(* Logix 5000 project; controller CLASE_1 Emulate 5570 rev 28.11; software revision 28.02; part 14 of 15 *)
(* tags used below, declared in another part *)
   FV_00_Intlk_Ok : BOOL;
   FV_00_Perm_Ok : BOOL;
   P_100_B_Intlk_OK : BOOL;
   PID_OUT_TK_200 : REAL;   // Esfuerzo de control Deberá ir direccionada a la salida analogica fisica
   PID_OUT_TK_300 : REAL;
   PPX_M_100 : P_DescList[1];
   PPX_M_200 : P_DescList[1];
   PPX_M_300 : P_DescList[1];
   PPX_P_100_B : P_DescList[1];
   PPX_P_200 : P_DescList[1];
   PPX_P_300 : P_DescList[1];
   PPX_Pump_100_A : P_DescList[1];
   Pump_100_A_Intlk_Ok : BOOL;

PROGRAM Equipos_TK_100   (* main routine MainProgram *)
VAR
   P_51A_B_Perm : P_Perm := (Inp_Perm01 := 1, Inp_Perm02 := 1, Inp_Perm03 := 1, Inp_Perm04 := 1, Inp_Perm05 := 1, Inp_Perm06 := 1, Inp_Perm07 := 1, Inp_Perm08 := 1, Inp_Perm09 := 1, Inp_Perm10 := 1, Inp_Perm11 := 1, Inp_Perm12 := 1, Inp_Perm13 := 1, Inp_Perm14 := 1, Inp_Perm15 := 1, Cfg_OKState := 2#1111_1111_1111_1111, Sts_Perm := 2#1111_1111_1111_1110);
   P_AIn_01 : P_AIn := (Inp_HiHiGate := 1, Inp_HiGate := 1, Inp_LoGate := 1, Inp_LoLoGate := 1, Inp_FailGate := 1, Cfg_SetTrack := 1, Cfg_PCmdClear := 1, Cfg_HiHiAckReqd := 1, Cfg_HiAckReqd := 1, Cfg_LoAckReqd := 1, Cfg_LoLoAckReqd := 1, Cfg_FailAckReqd := 1, Cfg_HiHiSeverity := 750, Cfg_HiSeverity := 500, Cfg_LoSeverity := 500, Cfg_LoLoSeverity := 750, Cfg_FailSeverity := 1000, Cfg_InpRawMax := 100.0, Cfg_PVEUMax := 100.0, Cfg_HiHiDB := 1.0, Cfg_HiDB := 1.0, Cfg_LoDB := 1.0, Cfg_LoLoDB := 1.0, Cfg_FailHiLim := 103.958336, Cfg_FailLoLim := -2.0833333, Cfg_FailDB := 0.41666666, PSet_HiHiLim := 1.5e+38, PSet_HiLim := 1.5e+38, PSet_LoLim := -1.5e+38, PSet_LoLoLim := -1.5e+38, OSet_HiHiLim := 1.5e+38, OSet_HiLim := 1.5e+38, OSet_LoLim := -1.5e+38, OSet_LoLoLim := -1.5e+38, Val_PVMinCapt := 1.5e+38, Val_PVMaxCapt := -1.5e+38, Val_PVEUMax := 100.0, Val_HiHiLim := 1.5e+38, Val_HiLim := 1.5e+38, Val_LoLim := -1.5e+38, Val_LoLoLim := -1.5e+38, Sts_InpPV := 1, Sts_Oper := 1, Ack_HiHi := 1, Ack_Hi := 1, Ack_Lo := 1, Ack_LoLo := 1, Ack_Fail := 1);
   P_AIn_02 : P_AIn := (Inp_HiHiGate := 1, Inp_HiGate := 1, Inp_LoGate := 1, Inp_LoLoGate := 1, Inp_FailGate := 1, Cfg_SetTrack := 1, Cfg_PCmdClear := 1, Cfg_HiHiAckReqd := 1, Cfg_HiAckReqd := 1, Cfg_LoAckReqd := 1, Cfg_LoLoAckReqd := 1, Cfg_FailAckReqd := 1, Cfg_HiHiSeverity := 750, Cfg_HiSeverity := 500, Cfg_LoSeverity := 500, Cfg_LoLoSeverity := 750, Cfg_FailSeverity := 1000, Cfg_InpRawMax := 100.0, Cfg_PVEUMax := 100.0, Cfg_HiHiDB := 1.0, Cfg_HiDB := 1.0, Cfg_LoDB := 1.0, Cfg_LoLoDB := 1.0, Cfg_FailHiLim := 103.958336, Cfg_FailLoLim := -2.0833333, Cfg_FailDB := 0.41666666, PSet_HiHiLim := 1.5e+38, PSet_HiLim := 1.5e+38, PSet_LoLim := -1.5e+38, PSet_LoLoLim := -1.5e+38, OSet_HiHiLim := 1.5e+38, OSet_HiLim := 1.5e+38, OSet_LoLim := -1.5e+38, OSet_LoLoLim := -1.5e+38, Val_PVMinCapt := 1.5e+38, Val_PVMaxCapt := -1.5e+38, Val_PVEUMax := 100.0, Val_HiHiLim := 1.5e+38, Val_HiLim := 1.5e+38, Val_LoLim := -1.5e+38, Val_LoLoLim := -1.5e+38, Sts_InpPV := 1, Sts_Oper := 1, Ack_HiHi := 1, Ack_Hi := 1, Ack_Lo := 1, Ack_LoLo := 1, Ack_Fail := 1);
   P_AIn_03 : P_AIn := (Inp_HiHiGate := 1, Inp_HiGate := 1, Inp_LoGate := 1, Inp_LoLoGate := 1, Inp_FailGate := 1, Cfg_SetTrack := 1, Cfg_PCmdClear := 1, Cfg_HiHiAckReqd := 1, Cfg_HiAckReqd := 1, Cfg_LoAckReqd := 1, Cfg_LoLoAckReqd := 1, Cfg_FailAckReqd := 1, Cfg_HiHiSeverity := 750, Cfg_HiSeverity := 500, Cfg_LoSeverity := 500, Cfg_LoLoSeverity := 750, Cfg_FailSeverity := 1000, Cfg_InpRawMax := 100.0, Cfg_PVEUMax := 100.0, Cfg_HiHiDB := 1.0, Cfg_HiDB := 1.0, Cfg_LoDB := 1.0, Cfg_LoLoDB := 1.0, Cfg_FailHiLim := 103.958336, Cfg_FailLoLim := -2.0833333, Cfg_FailDB := 0.41666666, PSet_HiHiLim := 1.5e+38, PSet_HiLim := 1.5e+38, PSet_LoLim := -1.5e+38, PSet_LoLoLim := -1.5e+38, OSet_HiHiLim := 1.5e+38, OSet_HiLim := 1.5e+38, OSet_LoLim := -1.5e+38, OSet_LoLoLim := -1.5e+38, Val_PVMinCapt := 1.5e+38, Val_PVMaxCapt := -1.5e+38, Val_PVEUMax := 100.0, Val_HiHiLim := 1.5e+38, Val_HiLim := 1.5e+38, Val_LoLim := -1.5e+38, Val_LoLoLim := -1.5e+38, Sts_InpPV := 1, Sts_Oper := 1, Ack_HiHi := 1, Ack_Hi := 1, Ack_Lo := 1, Ack_LoLo := 1, Ack_Fail := 1);
   P_AIn_04 : P_AIn := (Inp_HiHiGate := 1, Inp_HiGate := 1, Inp_LoGate := 1, Inp_LoLoGate := 1, Inp_FailGate := 1, Cfg_SetTrack := 1, Cfg_PCmdClear := 1, Cfg_HiHiAckReqd := 1, Cfg_HiAckReqd := 1, Cfg_LoAckReqd := 1, Cfg_LoLoAckReqd := 1, Cfg_FailAckReqd := 1, Cfg_HiHiSeverity := 750, Cfg_HiSeverity := 500, Cfg_LoSeverity := 500, Cfg_LoLoSeverity := 750, Cfg_FailSeverity := 1000, Cfg_InpRawMax := 100.0, Cfg_PVEUMax := 100.0, Cfg_HiHiDB := 1.0, Cfg_HiDB := 1.0, Cfg_LoDB := 1.0, Cfg_LoLoDB := 1.0, Cfg_FailHiLim := 103.958336, Cfg_FailLoLim := -2.0833333, Cfg_FailDB := 0.41666666, PSet_HiHiLim := 1.5e+38, PSet_HiLim := 1.5e+38, PSet_LoLim := -1.5e+38, PSet_LoLoLim := -1.5e+38, OSet_HiHiLim := 1.5e+38, OSet_HiLim := 1.5e+38, OSet_LoLim := -1.5e+38, OSet_LoLoLim := -1.5e+38, Val_PVMinCapt := 1.5e+38, Val_PVMaxCapt := -1.5e+38, Val_PVEUMax := 100.0, Val_HiHiLim := 1.5e+38, Val_HiLim := 1.5e+38, Val_LoLim := -1.5e+38, Val_LoLoLim := -1.5e+38, Sts_InpPV := 1, Sts_Oper := 1, Ack_HiHi := 1, Ack_Hi := 1, Ack_Lo := 1, Ack_LoLo := 1, Ack_Fail := 1);
   P_DIn_01 : P_DIn := (Inp_PV := 1, Inp_Target := 1, Inp_Gate := 1, Cfg_NormTextVis := 1, Cfg_PCmdClear := 1, Cfg_TgtDisagreeAckReqd := 1, Cfg_TgtDisagreeSeverity := 750, Ack_TgtDisagree := 1);
   P_DIn_02 : P_DIn := (Inp_PV := 1, Inp_Target := 1, Inp_Gate := 1, Cfg_NormTextVis := 1, Cfg_PCmdClear := 1, Cfg_TgtDisagreeAckReqd := 1, Cfg_TgtDisagreeSeverity := 750, Ack_TgtDisagree := 1);
   P_DIn_03 : P_DIn := (Inp_PV := 1, Inp_Target := 1, Inp_Gate := 1, Cfg_NormTextVis := 1, Cfg_PCmdClear := 1, Cfg_TgtDisagreeAckReqd := 1, Cfg_TgtDisagreeSeverity := 750, Ack_TgtDisagree := 1);
   P_Intlk_01 : P_Intlk := (Cfg_PCmdClear := 1, Sts_IntlkOK := 1, Sts_NBIntlkOK := 1);
   P_Intlk_02 : P_Intlk := (Cfg_PCmdClear := 1, Sts_IntlkOK := 1, Sts_NBIntlkOK := 1);
   P_Intlk_03 : P_Intlk := (Cfg_PCmdClear := 1, Sts_IntlkOK := 1, Sts_NBIntlkOK := 1);
   P_Intlk_04 : P_Intlk := (Cfg_PCmdClear := 1, Sts_IntlkOK := 1, Sts_NBIntlkOK := 1);
   P_Intlk_05 : P_Intlk := (Cfg_PCmdClear := 1, Sts_IntlkOK := 1, Sts_NBIntlkOK := 1);
   P_Intlk_06 : P_Intlk := (Cfg_PCmdClear := 1, Sts_IntlkOK := 1, Sts_NBIntlkOK := 1);
   P_Motor_01 : P_Motor := (Inp_PermOK := 1, Inp_NBPermOK := 1, Inp_IntlkOK := 1, Inp_NBIntlkOK := 1, Cfg_PCmdClear := 1, Cfg_ShedOnFailToStart := 1, Cfg_ShedOnIOFault := 1, Cfg_FailToStartAckReqd := 1, Cfg_FailToStopAckReqd := 1, Cfg_IntlkTripAckReqd := 1, Cfg_IOFaultAckReqd := 1, Cfg_FailToStartSeverity := 1000, Cfg_FailToStopSeverity := 1000, Cfg_IntlkTripSeverity := 500, Cfg_IOFaultSeverity := 1000, Cfg_SimFdbkT := 2, Cfg_FailToStartT := 10, Cfg_FailToStopT := 10, Sts_Stopped := 1, Sts_Oper := 1, Ack_FailToStart := 1, Ack_FailToStop := 1, Ack_IntlkTrip := 1, Ack_IOFault := 1);
   P_Motor_02 : P_Motor := (Inp_PermOK := 1, Inp_NBPermOK := 1, Inp_IntlkOK := 1, Inp_NBIntlkOK := 1, Cfg_PCmdClear := 1, Cfg_ShedOnFailToStart := 1, Cfg_ShedOnIOFault := 1, Cfg_FailToStartAckReqd := 1, Cfg_FailToStopAckReqd := 1, Cfg_IntlkTripAckReqd := 1, Cfg_IOFaultAckReqd := 1, Cfg_FailToStartSeverity := 1000, Cfg_FailToStopSeverity := 1000, Cfg_IntlkTripSeverity := 500, Cfg_IOFaultSeverity := 1000, Cfg_SimFdbkT := 2, Cfg_FailToStartT := 10, Cfg_FailToStopT := 10, Sts_Stopped := 1, Sts_Oper := 1, Ack_FailToStart := 1, Ack_FailToStop := 1, Ack_IntlkTrip := 1, Ack_IOFault := 1);
   P_Motor_03 : P_Motor := (Inp_PermOK := 1, Inp_NBPermOK := 1, Inp_IntlkOK := 1, Inp_NBIntlkOK := 1, Cfg_PCmdClear := 1, Cfg_ShedOnFailToStart := 1, Cfg_ShedOnIOFault := 1, Cfg_FailToStartAckReqd := 1, Cfg_FailToStopAckReqd := 1, Cfg_IntlkTripAckReqd := 1, Cfg_IOFaultAckReqd := 1, Cfg_FailToStartSeverity := 1000, Cfg_FailToStopSeverity := 1000, Cfg_IntlkTripSeverity := 500, Cfg_IOFaultSeverity := 1000, Cfg_SimFdbkT := 2, Cfg_FailToStartT := 10, Cfg_FailToStopT := 10, Sts_Stopped := 1, Sts_Oper := 1, Ack_FailToStart := 1, Ack_FailToStop := 1, Ack_IntlkTrip := 1, Ack_IOFault := 1);
   P_Perm_01 : P_Perm := (Inp_Perm00 := 1, Inp_Perm01 := 1, Inp_Perm02 := 1, Inp_Perm03 := 1, Inp_Perm04 := 1, Inp_Perm05 := 1, Inp_Perm06 := 1, Inp_Perm07 := 1, Inp_Perm08 := 1, Inp_Perm09 := 1, Inp_Perm10 := 1, Inp_Perm11 := 1, Inp_Perm12 := 1, Inp_Perm13 := 1, Inp_Perm14 := 1, Inp_Perm15 := 1, Cfg_OKState := 2#1111_1111_1111_1111, Sts_PermOK := 1, Sts_NBPermOK := 1, Sts_Perm := 2#1111_1111_1111_1111);
   P_Perm_02 : P_Perm := (Inp_Perm02 := 1, Inp_Perm03 := 1, Inp_Perm04 := 1, Inp_Perm05 := 1, Inp_Perm06 := 1, Inp_Perm07 := 1, Inp_Perm08 := 1, Inp_Perm09 := 1, Inp_Perm10 := 1, Inp_Perm11 := 1, Inp_Perm12 := 1, Inp_Perm13 := 1, Inp_Perm14 := 1, Inp_Perm15 := 1, Cfg_OKState := 2#1111_1111_1111_1111, Sts_Perm := 2#1111_1111_1111_1100);
   P_Perm_03 : P_Perm := (Inp_Perm00 := 1, Inp_Perm01 := 1, Inp_Perm02 := 1, Inp_Perm03 := 1, Inp_Perm04 := 1, Inp_Perm05 := 1, Inp_Perm06 := 1, Inp_Perm07 := 1, Inp_Perm08 := 1, Inp_Perm09 := 1, Inp_Perm10 := 1, Inp_Perm11 := 1, Inp_Perm12 := 1, Inp_Perm13 := 1, Inp_Perm14 := 1, Inp_Perm15 := 1, Cfg_OKState := 2#1111_1111_1111_1111, Sts_PermOK := 1, Sts_NBPermOK := 1, Sts_Perm := 2#1111_1111_1111_1111);
   P_Perm_04 : P_Perm := (Inp_Perm00 := 1, Inp_Perm01 := 1, Inp_Perm02 := 1, Inp_Perm03 := 1, Inp_Perm04 := 1, Inp_Perm05 := 1, Inp_Perm06 := 1, Inp_Perm07 := 1, Inp_Perm08 := 1, Inp_Perm09 := 1, Inp_Perm10 := 1, Inp_Perm11 := 1, Inp_Perm12 := 1, Inp_Perm13 := 1, Inp_Perm14 := 1, Inp_Perm15 := 1, Cfg_OKState := 2#1111_1111_1111_1111, Sts_PermOK := 1, Sts_NBPermOK := 1, Sts_Perm := 2#1111_1111_1111_1111);
   P_ValveC_01 : P_ValveC := (Inp_IntlkOK := 1, Inp_NBIntlkOK := 1, Cfg_ShedOnIOFault := 1, Cfg_SetTrack := 1, Cfg_LSFail := 1, Cfg_PCmdClear := 1, Cfg_ProgDefault := 1, Cfg_IntlkTripAckReqd := 1, Cfg_ActuatorFaultAckReqd := 1, Cfg_IOFaultAckReqd := 1, Cfg_IntlkTripSeverity := 500, Cfg_ActuatorFaultSeverity := 1000, Cfg_IOFaultSeverity := 1000, Cfg_MaxCV := 100.0, Cfg_MaxCVRoCInc := 10.0, Cfg_MaxCVRoCDec := 10.0, Cfg_CVEUMax := 100.0, Cfg_CVRawMin := 3277.0, Cfg_CVRawMax := 16384.0, Cfg_FdbkRawMax := 100.0, Cfg_CycleT := 10.0, Cfg_OpenRate := 1.0, Cfg_CloseRate := 1.0, Cfg_MaxOnT := 5.0, Cfg_MinOnT := 1.0, Val_CVEUMax := 100.0, Ack_IntlkTrip := 1, Ack_ActuatorFault := 1, Ack_IOFault := 1);
   P_ValveSO_01 : P_ValveSO := (Inp_PermOK := 1, Inp_NBPermOK := 1, Inp_IntlkOK := 1, Inp_NBIntlkOK := 1, Cfg_LSFail := 1, Cfg_PCmdClear := 1, Cfg_ShedOnFullStall := 1, Cfg_ShedOnTransitStall := 1, Cfg_ShedOnIOFault := 1, Cfg_FullStallAckReqd := 1, Cfg_TransitStallAckReqd := 1, Cfg_IntlkTripAckReqd := 1, Cfg_IOFaultAckReqd := 1, Cfg_FullStallSeverity := 1000, Cfg_TransitStallSeverity := 1000, Cfg_IntlkTripSeverity := 500, Cfg_IOFaultSeverity := 1000, Cfg_SimFdbkT := 2, Cfg_FullStallT := 5, Cfg_TransitStallT := 10, Ack_FullStall := 1, Ack_TransitStall := 1, Ack_IntlkTrip := 1, Ack_IOFault := 1);
   P_ValveSO_02 : P_ValveSO := (Inp_PermOK := 1, Inp_NBPermOK := 1, Inp_IntlkOK := 1, Inp_NBIntlkOK := 1, Cfg_LSFail := 1, Cfg_PCmdClear := 1, Cfg_ShedOnFullStall := 1, Cfg_ShedOnTransitStall := 1, Cfg_ShedOnIOFault := 1, Cfg_FullStallAckReqd := 1, Cfg_TransitStallAckReqd := 1, Cfg_IntlkTripAckReqd := 1, Cfg_IOFaultAckReqd := 1, Cfg_FullStallSeverity := 1000, Cfg_TransitStallSeverity := 1000, Cfg_IntlkTripSeverity := 500, Cfg_IOFaultSeverity := 1000, Cfg_SimFdbkT := 2, Cfg_FullStallT := 5, Cfg_TransitStallT := 10, Ack_FullStall := 1, Ack_TransitStall := 1, Ack_IntlkTrip := 1, Ack_IOFault := 1);
   P_VSD_01 : P_VSD := (Inp_Ready := 1, Inp_CommandDir := 1, Inp_ActualDir := 1, Inp_FwdPermOK := 1, Inp_FwdNBPermOK := 1, Inp_RevPermOK := 1, Inp_RevNBPermOK := 1, Inp_IntlkOK := 1, Inp_NBIntlkOK := 1, Cfg_SetTrack := 1, Cfg_PCmdClear := 1, Cfg_ShedOnFailToStart := 1, Cfg_ShedOnIOFault := 1, Cfg_FailToStartAckReqd := 1, Cfg_FailToStopAckReqd := 1, Cfg_IntlkTripAckReqd := 1, Cfg_DriveFaultAckReqd := 1, Cfg_IOFaultAckReqd := 1, Cfg_FailToStartSeverity := 1000, Cfg_FailToStopSeverity := 1000, Cfg_IntlkTripSeverity := 500, Cfg_DriveFaultSeverity := 1000, Cfg_IOFaultSeverity := 1000, Cfg_MaxSpdRef := 60.0, Cfg_SpeedRefRawMax := 32767.0, Cfg_SpeedRefEUMax := 130.0, Cfg_SpeedFdbkRawMax := 32767.0, Cfg_SpeedFdbkEUMax := 130.0, Cfg_InpDatalinkRawMax := 4095.0, Cfg_InpDatalinkEUMax := 409.5, Cfg_OutDatalinkMax := 100.0, Cfg_OutDatalinkRawMax := 4095.0, Cfg_OutDatalinkEUMax := 409.5, Cfg_SimRampT := 10, Cfg_FailToStartT := 15, Cfg_FailToStopT := 15, Cfg_ResetPulseT := 2, Val_SpeedRefEUMax := 130.0, Val_SpeedFdbkEUMax := 130.0, Ack_FailToStart := 1, Ack_FailToStop := 1, Ack_IntlkTrip := 1, Ack_DriveFault := 1, Ack_IOFault := 1);
END_VAR

ROUTINE _00_Valvulas   (* function block diagram *)
   SHEET 1   // FV_100
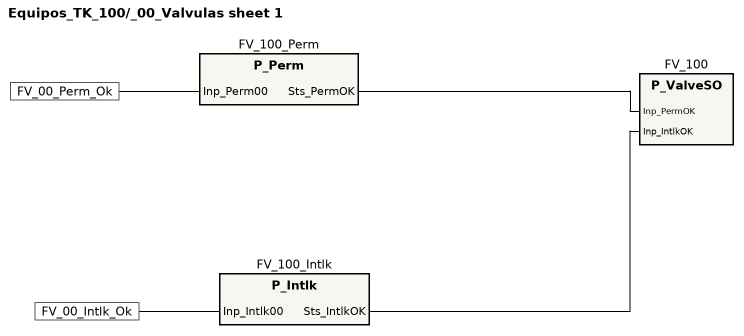
   FV_100_Perm : P_Perm(Inp_Perm00 := FV_00_Perm_Ok);
   FV_100_Intlk : P_Intlk(Inp_Intlk00 := FV_00_Intlk_Ok);
   FV_100 : P_ValveSO(Inp_PermOK := FV_100_Perm.Sts_PermOK, Inp_IntlkOK := FV_100_Intlk.Sts_IntlkOK);
END_ROUTINE

ROUTINE _02_Motores   (* function block diagram *)
   SHEET 1   // Pump_100_A
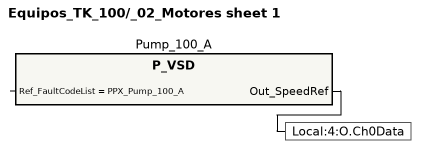
   Pump_100_A : P_VSD(Ref_FaultCodeList := PPX_Pump_100_A);
   Local:4:O.Ch0Data := Pump_100_A.Out_SpeedRef;
   SHEET 2   // Triturador_M_100
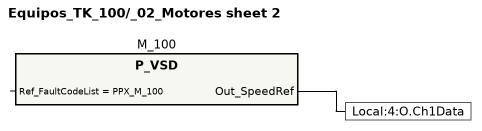
   M_100 : P_VSD(Ref_FaultCodeList := PPX_M_100);
   Local:4:O.Ch1Data := M_100.Out_SpeedRef;
END_ROUTINE

ROUTINE _03_Entrada_Digital   (* function block diagram *)
   SHEET 1
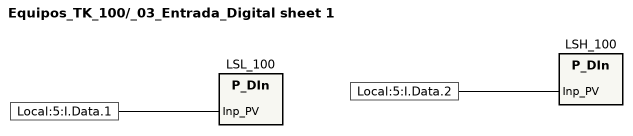
   LSL_100 : P_DIn(Inp_PV := Local:5:I.Data.1);
   LSH_100 : P_DIn(Inp_PV := Local:5:I.Data.2);
END_ROUTINE

ROUTINE Condiciones   (* ladder *)
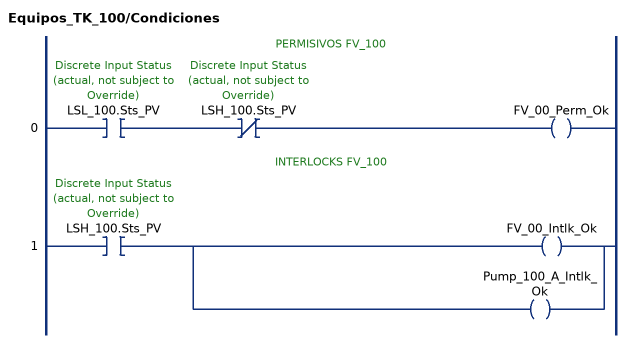
   // PERMISIVOS FV_100
   0: XIC(LSL_100.Sts_PV)XIO(LSH_100.Sts_PV)OTE(FV_00_Perm_Ok);
   // INTERLOCKS FV_100
   1: XIC(LSH_100.Sts_PV)[OTE(FV_00_Intlk_Ok) ,OTE(Pump_100_A_Intlk_Ok) ];
END_ROUTINE

ROUTINE MainProgram   (* ladder *)
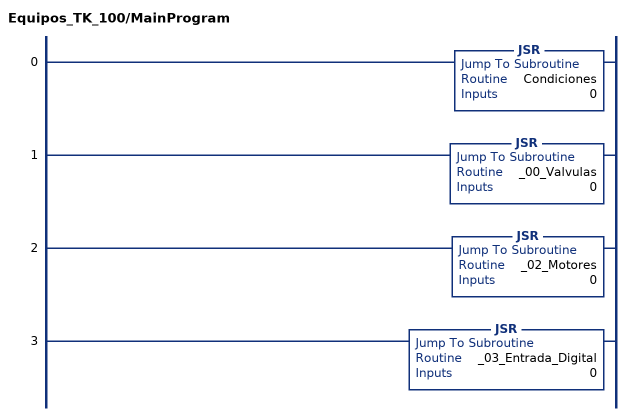
   0: JSR(Condiciones,0);
   1: JSR(_00_Valvulas,0);
   2: JSR(_02_Motores,0);
   3: JSR(_03_Entrada_Digital,0);
END_ROUTINE
END_PROGRAM

PROGRAM Equipos_TK_200   (* main routine Main *)
VAR
   P_AIn_01 : P_AIn := (Inp_HiHiGate := 1, Inp_HiGate := 1, Inp_LoGate := 1, Inp_LoLoGate := 1, Inp_FailGate := 1, Cfg_SetTrack := 1, Cfg_PCmdClear := 1, Cfg_HiHiAckReqd := 1, Cfg_HiAckReqd := 1, Cfg_LoAckReqd := 1, Cfg_LoLoAckReqd := 1, Cfg_FailAckReqd := 1, Cfg_HiHiSeverity := 750, Cfg_HiSeverity := 500, Cfg_LoSeverity := 500, Cfg_LoLoSeverity := 750, Cfg_FailSeverity := 1000, Cfg_InpRawMax := 100.0, Cfg_PVEUMax := 100.0, Cfg_HiHiDB := 1.0, Cfg_HiDB := 1.0, Cfg_LoDB := 1.0, Cfg_LoLoDB := 1.0, Cfg_FailHiLim := 103.958336, Cfg_FailLoLim := -2.0833333, Cfg_FailDB := 0.41666666, PSet_HiHiLim := 1.5e+38, PSet_HiLim := 1.5e+38, PSet_LoLim := -1.5e+38, PSet_LoLoLim := -1.5e+38, OSet_HiHiLim := 1.5e+38, OSet_HiLim := 1.5e+38, OSet_LoLim := -1.5e+38, OSet_LoLoLim := -1.5e+38, Val_PVMinCapt := 1.5e+38, Val_PVMaxCapt := -1.5e+38, Val_PVEUMax := 100.0, Val_HiHiLim := 1.5e+38, Val_HiLim := 1.5e+38, Val_LoLim := -1.5e+38, Val_LoLoLim := -1.5e+38, Sts_InpPV := 1, Sts_Oper := 1, Ack_HiHi := 1, Ack_Hi := 1, Ack_Lo := 1, Ack_LoLo := 1, Ack_Fail := 1);
   P_DIn_01 : P_DIn := (Inp_PV := 1, Inp_Target := 1, Inp_Gate := 1, Cfg_NormTextVis := 1, Cfg_PCmdClear := 1, Cfg_TgtDisagreeAckReqd := 1, Cfg_TgtDisagreeSeverity := 750, Ack_TgtDisagree := 1);
   P_Intlk_01 : P_Intlk := (Cfg_PCmdClear := 1, Sts_IntlkOK := 1, Sts_NBIntlkOK := 1);
   P_Intlk_02 : P_Intlk := (Cfg_PCmdClear := 1, Sts_IntlkOK := 1, Sts_NBIntlkOK := 1);
   P_Perm_01 : P_Perm := (Inp_Perm00 := 1, Inp_Perm01 := 1, Inp_Perm02 := 1, Inp_Perm03 := 1, Inp_Perm04 := 1, Inp_Perm05 := 1, Inp_Perm06 := 1, Inp_Perm07 := 1, Inp_Perm08 := 1, Inp_Perm09 := 1, Inp_Perm10 := 1, Inp_Perm11 := 1, Inp_Perm12 := 1, Inp_Perm13 := 1, Inp_Perm14 := 1, Inp_Perm15 := 1, Cfg_OKState := 2#1111_1111_1111_1111, Sts_PermOK := 1, Sts_NBPermOK := 1, Sts_Perm := 2#1111_1111_1111_1111);
   P_ValveSO_01 : P_ValveSO := (Inp_PermOK := 1, Inp_NBPermOK := 1, Inp_IntlkOK := 1, Inp_NBIntlkOK := 1, Cfg_LSFail := 1, Cfg_PCmdClear := 1, Cfg_ShedOnFullStall := 1, Cfg_ShedOnTransitStall := 1, Cfg_ShedOnIOFault := 1, Cfg_FullStallAckReqd := 1, Cfg_TransitStallAckReqd := 1, Cfg_IntlkTripAckReqd := 1, Cfg_IOFaultAckReqd := 1, Cfg_FullStallSeverity := 1000, Cfg_TransitStallSeverity := 1000, Cfg_IntlkTripSeverity := 500, Cfg_IOFaultSeverity := 1000, Cfg_SimFdbkT := 2, Cfg_FullStallT := 5, Cfg_TransitStallT := 10, Ack_FullStall := 1, Ack_TransitStall := 1, Ack_IntlkTrip := 1, Ack_IOFault := 1);
   P_VSD_01 : P_VSD := (Inp_Ready := 1, Inp_CommandDir := 1, Inp_ActualDir := 1, Inp_FwdPermOK := 1, Inp_FwdNBPermOK := 1, Inp_RevPermOK := 1, Inp_RevNBPermOK := 1, Inp_IntlkOK := 1, Inp_NBIntlkOK := 1, Cfg_SetTrack := 1, Cfg_PCmdClear := 1, Cfg_ShedOnFailToStart := 1, Cfg_ShedOnIOFault := 1, Cfg_FailToStartAckReqd := 1, Cfg_FailToStopAckReqd := 1, Cfg_IntlkTripAckReqd := 1, Cfg_DriveFaultAckReqd := 1, Cfg_IOFaultAckReqd := 1, Cfg_FailToStartSeverity := 1000, Cfg_FailToStopSeverity := 1000, Cfg_IntlkTripSeverity := 500, Cfg_DriveFaultSeverity := 1000, Cfg_IOFaultSeverity := 1000, Cfg_MaxSpdRef := 60.0, Cfg_SpeedRefRawMax := 32767.0, Cfg_SpeedRefEUMax := 130.0, Cfg_SpeedFdbkRawMax := 32767.0, Cfg_SpeedFdbkEUMax := 130.0, Cfg_InpDatalinkRawMax := 4095.0, Cfg_InpDatalinkEUMax := 409.5, Cfg_OutDatalinkMax := 100.0, Cfg_OutDatalinkRawMax := 4095.0, Cfg_OutDatalinkEUMax := 409.5, Cfg_SimRampT := 10, Cfg_FailToStartT := 15, Cfg_FailToStopT := 15, Cfg_ResetPulseT := 2, Val_SpeedRefEUMax := 130.0, Val_SpeedFdbkEUMax := 130.0, Ack_FailToStart := 1, Ack_FailToStop := 1, Ack_IntlkTrip := 1, Ack_DriveFault := 1, Ack_IOFault := 1);
END_VAR

ROUTINE _00_Valvulas   (* function block diagram *)
   SHEET 1   // TCV_200
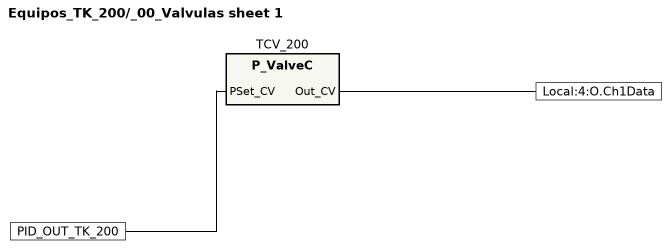
   TCV_200 : P_ValveC(PSet_CV := PID_OUT_TK_200);
   Local:4:O.Ch1Data := TCV_200.Out_CV;
END_ROUTINE

ROUTINE _01_Entrada_Analogica   (* function block diagram *)
   SHEET 1
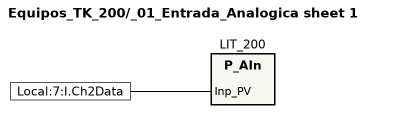
   LIT_200 : P_AIn(Inp_PV := Local:7:I.Ch2Data);
END_ROUTINE

ROUTINE _02_Motores   (* function block diagram *)
   SHEET 1   // P_100_B
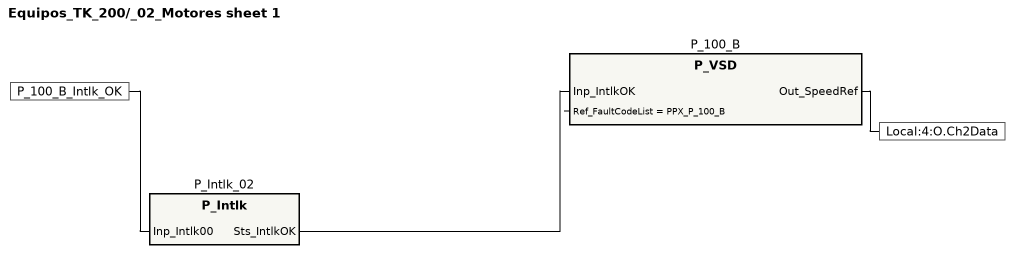
   P_Intlk_02 : P_Intlk(Inp_Intlk00 := P_100_B_Intlk_OK);
   P_100_B : P_VSD(Inp_IntlkOK := P_Intlk_02.Sts_IntlkOK, Ref_FaultCodeList := PPX_P_100_B);
   Local:4:O.Ch2Data := P_100_B.Out_SpeedRef;
   SHEET 2   // M_200
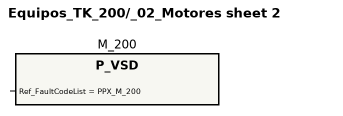
   M_200 : P_VSD(Ref_FaultCodeList := PPX_M_200);
END_ROUTINE

ROUTINE _03_Entradas_Digitales   (* function block diagram *)
   SHEET 1   // FSL_200
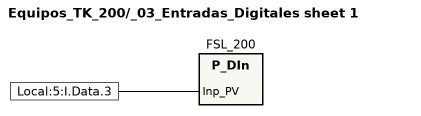
   FSL_200 : P_DIn(Inp_PV := Local:5:I.Data.3);
END_ROUTINE

ROUTINE Condiciones   (* ladder *)
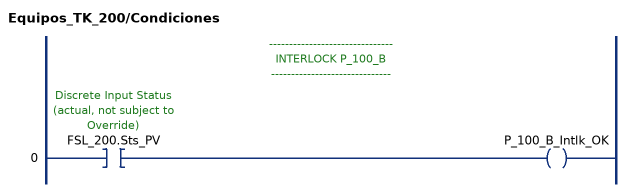
   // -------------------------------
   // INTERLOCK P_100_B
   // ------------------------------
   0: XIC(FSL_200.Sts_PV)OTE(P_100_B_Intlk_OK);
END_ROUTINE

ROUTINE Main   (* ladder *)
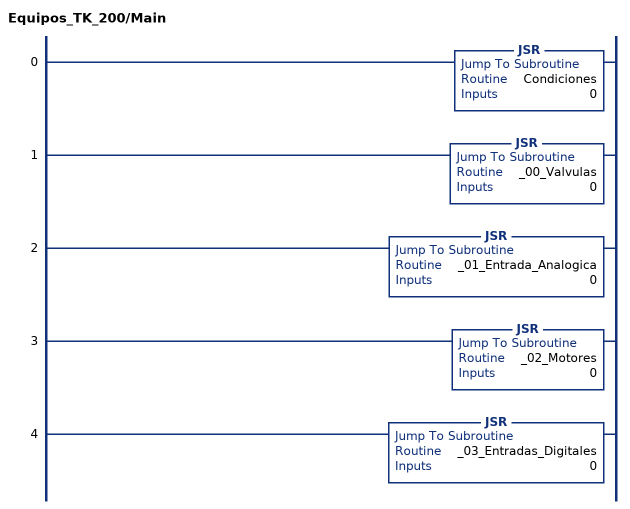
   0: JSR(Condiciones,0);
   1: JSR(_00_Valvulas,0);
   2: JSR(_01_Entrada_Analogica,0);
   3: JSR(_02_Motores,0);
   4: JSR(_03_Entradas_Digitales,0);
END_ROUTINE
END_PROGRAM

PROGRAM Equipos_TK_300   (* main routine Main *)
VAR
   P_AIn_01 : P_AIn := (Inp_HiHiGate := 1, Inp_HiGate := 1, Inp_LoGate := 1, Inp_LoLoGate := 1, Inp_FailGate := 1, Cfg_SetTrack := 1, Cfg_PCmdClear := 1, Cfg_HiHiAckReqd := 1, Cfg_HiAckReqd := 1, Cfg_LoAckReqd := 1, Cfg_LoLoAckReqd := 1, Cfg_FailAckReqd := 1, Cfg_HiHiSeverity := 750, Cfg_HiSeverity := 500, Cfg_LoSeverity := 500, Cfg_LoLoSeverity := 750, Cfg_FailSeverity := 1000, Cfg_InpRawMax := 100.0, Cfg_PVEUMax := 100.0, Cfg_HiHiDB := 1.0, Cfg_HiDB := 1.0, Cfg_LoDB := 1.0, Cfg_LoLoDB := 1.0, Cfg_FailHiLim := 103.958336, Cfg_FailLoLim := -2.0833333, Cfg_FailDB := 0.41666666, PSet_HiHiLim := 1.5e+38, PSet_HiLim := 1.5e+38, PSet_LoLim := -1.5e+38, PSet_LoLoLim := -1.5e+38, OSet_HiHiLim := 1.5e+38, OSet_HiLim := 1.5e+38, OSet_LoLim := -1.5e+38, OSet_LoLoLim := -1.5e+38, Val_PVMinCapt := 1.5e+38, Val_PVMaxCapt := -1.5e+38, Val_PVEUMax := 100.0, Val_HiHiLim := 1.5e+38, Val_HiLim := 1.5e+38, Val_LoLim := -1.5e+38, Val_LoLoLim := -1.5e+38, Sts_InpPV := 1, Sts_Oper := 1, Ack_HiHi := 1, Ack_Hi := 1, Ack_Lo := 1, Ack_LoLo := 1, Ack_Fail := 1);
   P_DIn_01 : P_DIn := (Inp_PV := 1, Inp_Target := 1, Inp_Gate := 1, Cfg_NormTextVis := 1, Cfg_PCmdClear := 1, Cfg_TgtDisagreeAckReqd := 1, Cfg_TgtDisagreeSeverity := 750, Ack_TgtDisagree := 1);
   P_Intlk_01 : P_Intlk := (Cfg_PCmdClear := 1, Sts_IntlkOK := 1, Sts_NBIntlkOK := 1);
   P_Perm_01 : P_Perm := (Inp_Perm00 := 1, Inp_Perm01 := 1, Inp_Perm02 := 1, Inp_Perm03 := 1, Inp_Perm04 := 1, Inp_Perm05 := 1, Inp_Perm06 := 1, Inp_Perm07 := 1, Inp_Perm08 := 1, Inp_Perm09 := 1, Inp_Perm10 := 1, Inp_Perm11 := 1, Inp_Perm12 := 1, Inp_Perm13 := 1, Inp_Perm14 := 1, Inp_Perm15 := 1, Cfg_OKState := 2#1111_1111_1111_1111, Sts_PermOK := 1, Sts_NBPermOK := 1, Sts_Perm := 2#1111_1111_1111_1111);
   P_ValveSO_01 : P_ValveSO := (Inp_PermOK := 1, Inp_NBPermOK := 1, Inp_IntlkOK := 1, Inp_NBIntlkOK := 1, Cfg_LSFail := 1, Cfg_PCmdClear := 1, Cfg_ShedOnFullStall := 1, Cfg_ShedOnTransitStall := 1, Cfg_ShedOnIOFault := 1, Cfg_FullStallAckReqd := 1, Cfg_TransitStallAckReqd := 1, Cfg_IntlkTripAckReqd := 1, Cfg_IOFaultAckReqd := 1, Cfg_FullStallSeverity := 1000, Cfg_TransitStallSeverity := 1000, Cfg_IntlkTripSeverity := 500, Cfg_IOFaultSeverity := 1000, Cfg_SimFdbkT := 2, Cfg_FullStallT := 5, Cfg_TransitStallT := 10, Ack_FullStall := 1, Ack_TransitStall := 1, Ack_IntlkTrip := 1, Ack_IOFault := 1);
   P_VSD_01 : P_VSD := (Inp_Ready := 1, Inp_CommandDir := 1, Inp_ActualDir := 1, Inp_FwdPermOK := 1, Inp_FwdNBPermOK := 1, Inp_RevPermOK := 1, Inp_RevNBPermOK := 1, Inp_IntlkOK := 1, Inp_NBIntlkOK := 1, Cfg_SetTrack := 1, Cfg_PCmdClear := 1, Cfg_ShedOnFailToStart := 1, Cfg_ShedOnIOFault := 1, Cfg_FailToStartAckReqd := 1, Cfg_FailToStopAckReqd := 1, Cfg_IntlkTripAckReqd := 1, Cfg_DriveFaultAckReqd := 1, Cfg_IOFaultAckReqd := 1, Cfg_FailToStartSeverity := 1000, Cfg_FailToStopSeverity := 1000, Cfg_IntlkTripSeverity := 500, Cfg_DriveFaultSeverity := 1000, Cfg_IOFaultSeverity := 1000, Cfg_MaxSpdRef := 60.0, Cfg_SpeedRefRawMax := 32767.0, Cfg_SpeedRefEUMax := 130.0, Cfg_SpeedFdbkRawMax := 32767.0, Cfg_SpeedFdbkEUMax := 130.0, Cfg_InpDatalinkRawMax := 4095.0, Cfg_InpDatalinkEUMax := 409.5, Cfg_OutDatalinkMax := 100.0, Cfg_OutDatalinkRawMax := 4095.0, Cfg_OutDatalinkEUMax := 409.5, Cfg_SimRampT := 10, Cfg_FailToStartT := 15, Cfg_FailToStopT := 15, Cfg_ResetPulseT := 2, Val_SpeedRefEUMax := 130.0, Val_SpeedFdbkEUMax := 130.0, Ack_FailToStart := 1, Ack_FailToStop := 1, Ack_IntlkTrip := 1, Ack_DriveFault := 1, Ack_IOFault := 1);
   P_VSD_02 : P_VSD := (Inp_Ready := 1, Inp_CommandDir := 1, Inp_ActualDir := 1, Inp_FwdPermOK := 1, Inp_FwdNBPermOK := 1, Inp_RevPermOK := 1, Inp_RevNBPermOK := 1, Inp_IntlkOK := 1, Inp_NBIntlkOK := 1, Cfg_SetTrack := 1, Cfg_PCmdClear := 1, Cfg_ShedOnFailToStart := 1, Cfg_ShedOnIOFault := 1, Cfg_FailToStartAckReqd := 1, Cfg_FailToStopAckReqd := 1, Cfg_IntlkTripAckReqd := 1, Cfg_DriveFaultAckReqd := 1, Cfg_IOFaultAckReqd := 1, Cfg_FailToStartSeverity := 1000, Cfg_FailToStopSeverity := 1000, Cfg_IntlkTripSeverity := 500, Cfg_DriveFaultSeverity := 1000, Cfg_IOFaultSeverity := 1000, Cfg_MaxSpdRef := 60.0, Cfg_SpeedRefRawMax := 32767.0, Cfg_SpeedRefEUMax := 130.0, Cfg_SpeedFdbkRawMax := 32767.0, Cfg_SpeedFdbkEUMax := 130.0, Cfg_InpDatalinkRawMax := 4095.0, Cfg_InpDatalinkEUMax := 409.5, Cfg_OutDatalinkMax := 100.0, Cfg_OutDatalinkRawMax := 4095.0, Cfg_OutDatalinkEUMax := 409.5, Cfg_SimRampT := 10, Cfg_FailToStartT := 15, Cfg_FailToStopT := 15, Cfg_ResetPulseT := 2, Val_SpeedRefEUMax := 130.0, Val_SpeedFdbkEUMax := 130.0, Ack_FailToStart := 1, Ack_FailToStop := 1, Ack_IntlkTrip := 1, Ack_DriveFault := 1, Ack_IOFault := 1);
END_VAR

ROUTINE _00_Valvulas   (* function block diagram *)
   SHEET 1   // TCV_200
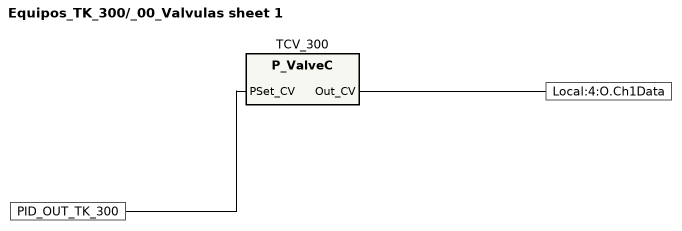
   TCV_300 : P_ValveC(PSet_CV := PID_OUT_TK_300);
   Local:4:O.Ch1Data := TCV_300.Out_CV;
END_ROUTINE

ROUTINE _01_Entrada_Analogica   (* function block diagram *)
   SHEET 1
END_ROUTINE

ROUTINE _02_Motores   (* function block diagram *)
   SHEET 1   // P_200
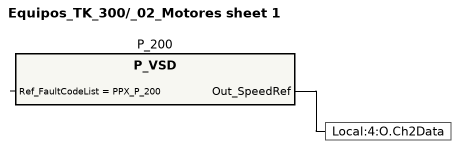
   P_200 : P_VSD(Ref_FaultCodeList := PPX_P_200);
   Local:4:O.Ch2Data := P_200.Out_SpeedRef;
   SHEET 2   // M_300
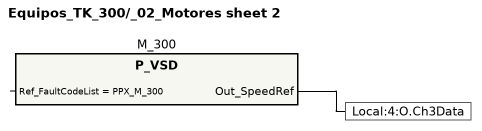
   M_300 : P_VSD(Ref_FaultCodeList := PPX_M_300);
   Local:4:O.Ch3Data := M_300.Out_SpeedRef;
   SHEET 3   // P_300
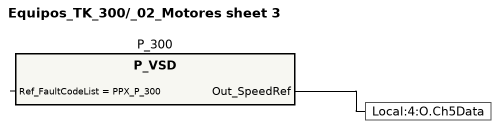
   P_300 : P_VSD(Ref_FaultCodeList := PPX_P_300);
   Local:4:O.Ch5Data := P_300.Out_SpeedRef;
END_ROUTINE

ROUTINE Condiciones   (* ladder *)
END_ROUTINE

ROUTINE Main   (* ladder *)
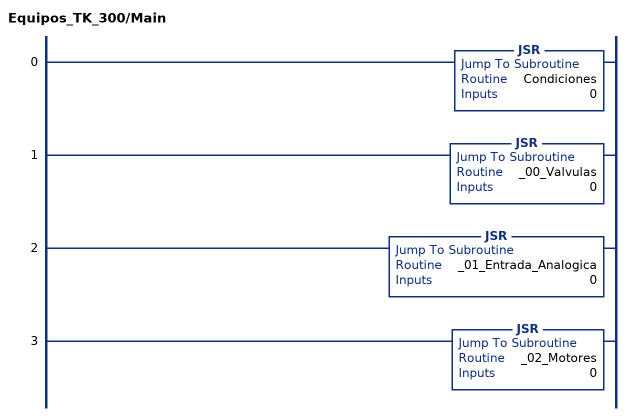
   0: JSR(Condiciones,0);
   1: JSR(_00_Valvulas,0);
   2: JSR(_01_Entrada_Analogica,0);
   3: JSR(_02_Motores,0);
END_ROUTINE
END_PROGRAM
